FUNCTION_BLOCK LargeSortingConveyor EXTENDS Conveyor
VAR_INPUT
END_VAR
VAR_OUTPUT
END_VAR
VAR
	m_rampPusherStart : MonostableCylinder;
	m_rampPusherMid : MonostableCylinder;
	m_Switch : Switch;
	
	m_presenceSensorStart : PresenceSensor;
	m_opticalSensorStart : OpticalSensor;
	m_opticalSensorMid : OpticalSensor;
	m_opticalSensorEnd : OpticalSensor;
	m_inductiveSensorStart : InductiveSensor;
	m_inductiveSensorMid : InductiveSensor;
	
	m_rampStart : Ramp;
	m_rampMiddle : Ramp;
	m_rampEnd : Ramp;
END_VAR

PROPERTY LightWPAtEnd : BOOL
GET
LightWPAtEnd := m_opticalSensorEnd.Value;
END_GET
END_PROPERTY

PROPERTY LightWPAtMid : BOOL
GET
LightWPAtMid := m_opticalSensorMid.Value;
END_GET
END_PROPERTY

PROPERTY LightWPAtStart : BOOL
GET
LightWPAtStart := m_opticalSensorStart.Value;
END_GET
END_PROPERTY

PROPERTY MetalWPAtMid : BOOL
GET
MetalWPAtMid := m_inductiveSensorMid.Value;
END_GET
END_PROPERTY

PROPERTY MetalWPAtStart : BOOL
GET
MetalWPAtStart := m_inductiveSensorStart.Value;
END_GET
END_PROPERTY

METHOD METH_Ramp1Pusher_Extend : BOOL
VAR_INPUT
END_VAR
m_rampPusherStart.METH_Extend();
END_METHOD

METHOD METH_Ramp1Pusher_Retract : BOOL
VAR_INPUT
END_VAR
m_rampPusherStart.METH_Retract();
END_METHOD

METHOD METH_Ramp2Pusher_Extend : BOOL
VAR_INPUT
END_VAR
m_rampPusherMid.METH_Extend();
END_METHOD

METHOD METH_Ramp2Pusher_Retract : BOOL
VAR_INPUT
END_VAR
m_rampPusherMid.METH_Retract();
END_METHOD

METHOD METH_Switch_Extend : BOOL
VAR_INPUT
END_VAR
m_Switch.METH_Extend();
END_METHOD

METHOD METH_Switch_Retract : BOOL
VAR_INPUT
END_VAR
m_Switch.METH_Retract();
END_METHOD

PROPERTY WPAtRampEnd : BOOL
GET
WPAtRampEnd := m_rampEnd.m_presenceSensorRampFull.Value;
END_GET
END_PROPERTY

PROPERTY WPAtRampMiddle : BOOL
GET
WPAtRampMiddle := m_rampMiddle.m_presenceSensorRampFull.Value;
END_GET
END_PROPERTY

PROPERTY WPAtRampStart : BOOL
GET
WPAtRampStart := m_rampStart.m_presenceSensorRampFull.Value;
END_GET
END_PROPERTY

PROPERTY WPAtStart : BOOL
GET
WPAtStart := m_presenceSensorStart.Value;
END_GET
END_PROPERTY

END_FUNCTION_BLOCK

(* stored: Version 1.1.0.1, ProductVersion 3.1.4024.9
   POU LargeSortingConveyor: Id {98c8a6c0-62a5-45da-9881-5971e7ae3c1a}, SpecialFunc None
   Folder Methods: Id {8ff7c17f-a5be-4131-85e0-cba796ee2f03}
   Folder Properties: Id {e064af6c-3a9d-4627-9c8b-8ce1c74285e0}
   Property LightWPAtEnd: Id {cbaaad75-a50b-4b75-a2ff-fb1ae4661bb2}
   Get Get: Id {789630a6-5abe-4f13-aa23-24a039dbdb39}
   Property LightWPAtMid: Id {c0691c77-34d2-4967-8f46-59f09c92b70f}
   Get Get: Id {f69fdf35-c4f0-469e-b359-271887fe662f}
   Property LightWPAtStart: Id {02423b6b-5a6d-44c0-9127-6a1044dfca19}
   Get Get: Id {47fea6c9-28f5-4489-bbd4-19a34fdb0e90}
   Property MetalWPAtMid: Id {08c93616-276a-4a9b-b348-c79ee62f39e2}
   Get Get: Id {06880b0f-ee17-4071-8e67-d014fff530de}
   Property MetalWPAtStart: Id {e1aff909-30a2-4e4a-9ef9-73515ae9b1d2}
   Get Get: Id {48d05e8a-cdb2-4a1f-9865-6d8e1a5e089b}
   Method METH_Ramp1Pusher_Extend: Id {db7aa33f-f817-42d9-b049-c5d7e89872a1}
   Method METH_Ramp1Pusher_Retract: Id {c93f0b37-9b41-472a-b2c4-919b8b97d70b}
   Method METH_Ramp2Pusher_Extend: Id {df550365-0219-49f9-a5e0-0d1ae07e1214}
   Method METH_Ramp2Pusher_Retract: Id {1e9a7802-1fbd-4d97-b3d8-c1d68e075485}
   Method METH_Switch_Extend: Id {888745d1-31ee-4883-a19a-52870fa1d2f8}
   Method METH_Switch_Retract: Id {0f674d0f-f954-4aea-8ce3-8203b48f6fbf}
   Property WPAtRampEnd: Id {72a736d8-8702-43de-bb34-0f294d57dfc1}
   Get Get: Id {6460b0d0-d378-4057-b1e0-1d22fb0c7f9b}
   Property WPAtRampMiddle: Id {eccfe64b-6438-4d2d-9171-848fed8750eb}
   Get Get: Id {44cef745-a3c0-4a76-b161-64da40a9d405}
   Property WPAtRampStart: Id {bf2003e6-aa99-498f-a066-ac1cd0c836c1}
   Get Get: Id {b86e42f8-f188-4e5d-9d15-696f18c9fdc3}
   Property WPAtStart: Id {012c0511-df99-49a9-9f7e-84c3f72bc727}
   Get Get: Id {355c7cca-f0d7-4aff-9909-5062632b7688} *)
